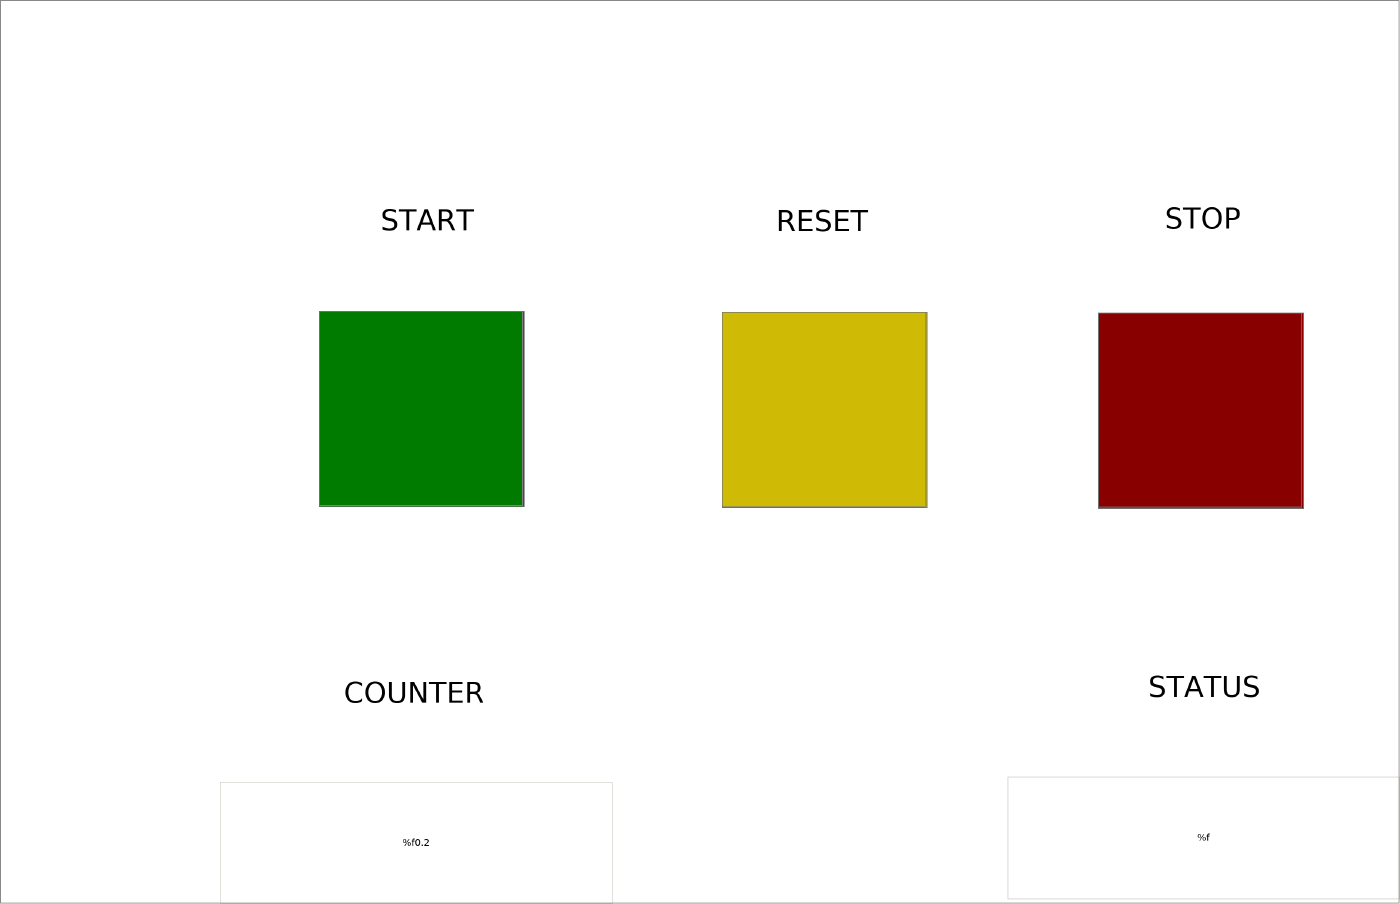
VISUALIZATION Visualization_Start_Screen  // 1637x1058
    Button (373,364 240x229), colour toggle: FIO.bEbStart
        OnMouseClick: toggle FIO.bEbStart
    Button (1284,366 240x229), colour toggle: FIO.bEbStopLight
        toggle FIO.bEbStop
        OnMouseClick: toggle FIO.bEbStop
    Textfield (257,915 459x143), "%f0.2", text variable: FIO.iEbCounter
    Textfield (1178,909 459x143), "%f", text variable: FIO.bEbAuto
    Textfield (399,230 201x55), "START"
    Textfield (1306,228 201x55), "STOP"
    Textfield (384,783 201x55), "COUNTER"
    Textfield (1308,776 201x55), "STATUS"
    Button (844,365 240x229), colour toggle: FIO.bEbReset
        OnMouseClick: toggle FIO.bEbReset
    Textfield (861,231 201x55), "RESET"
END_VISUALIZATION

(* stored: Version 1.1.0.1, ProductVersion 3.1.4024.3
   Visu Visualization_Start_Screen: Id {322834ea-a936-4e2a-a163-91e928bf6ab4} *)
